{attribute 'qualified_only'}
VAR_GLOBAL CONSTANT
	LABEL_LEN : USINT := 40;
	MESSAGE_LEN : USINT := 255;
END_VAR

(* stored: Version 1.1.0.1, ProductVersion 3.1.4024.12
   GVL Param_Error: Id {9d65e756-28ca-4528-a0e1-59b8d97cae72} *)
